(* Logix 5000 project; controller EsteiraSeletoraParte3 vendor 1 type 14 code 89 rev 20.11; software revision 20.05 *)

TASK MainTask (continuous, watchdog 500 ms) : MainProgram

MODULES
   Controller : vendor 1 type 14 code 89 (CompactLogixL23E_QBFC1_Controller 0, rev 20.11)
      LocalENB : vendor 1 type 12 code 191 (CompactLogixL23E_QBFC1_Ethernet 1, rev 20.11)
      Local : CompactBus (CompactVirtualAdapter 3, rev 20.11)
         Discrete_Inputs : vendor 1 type 7 code 320 (Compact 1, rev 3.1, Input RPI 20 ms)
         Discrete_Outputs : vendor 1 type 7 code 322 (Compact 2, rev 3.1, Output RPI 20 ms)
         Analog_IO : vendor 1 type 10 code 120 (Compact 3, rev 1.1, Output RPI 80 ms)
         Counters : vendor 1 type 109 code 70 (Compact 4, rev 1.1, Output RPI 20 ms)
END_MODULES

PROGRAM MainProgram   (* main routine MainRoutine *)
VAR
   AcionaEstacao1 : BOOL;
   AcionaEstacao2 : BOOL;
   AcionaEstacao3 : BOOL;
   EntroEstacao1 : BOOL;
   EntroEstacao2 : BOOL;
   EntroEstacao3 : BOOL;
   EsperaParaParar : TIMER;
   Estacao1 : BOOL;
   Estacao2 : BOOL;
   Estacao3 : BOOL;
   MotorEsteira : ALIAS FOR Local:2:O.Data.9;
   SensorEstacao1 : ALIAS FOR Local:1:I.Data.8;
   SensorEstacao2 : ALIAS FOR Local:1:I.Data.9;
   SensorEstacao3 : ALIAS FOR Local:1:I.Data.10;
   SistemaLigado : BOOL;
   StartStop : ALIAS FOR Local:1:I.Data.3;
   TrabalhandoEm1 : TIMER := (PRE := 1000);
   TrabalhandoEm2 : TIMER := (PRE := 2000);
   TrabalhandoEm3 : TIMER := (PRE := 3000);
END_VAR

ROUTINE MainRoutine   (* ladder *)
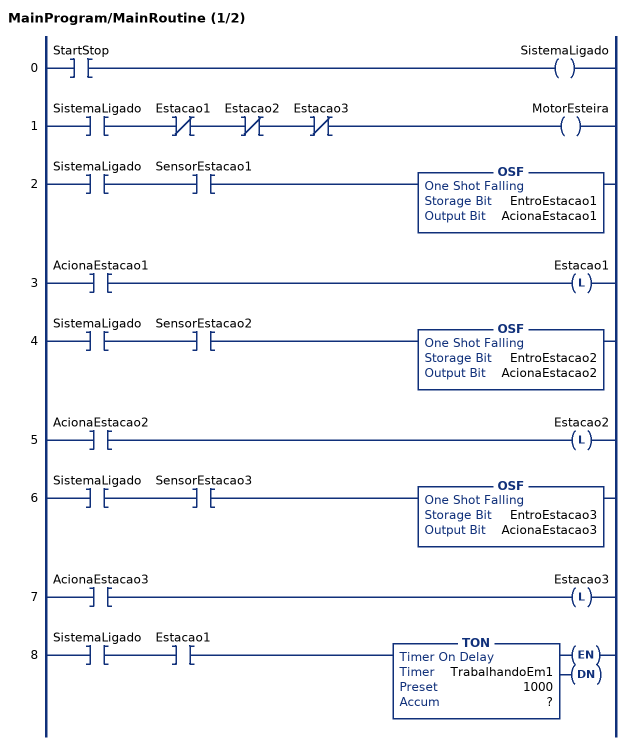
   0: XIC(StartStop)OTE(SistemaLigado);
   1: XIC(SistemaLigado)XIO(Estacao1)XIO(Estacao2)XIO(Estacao3)OTE(MotorEsteira);
   2: XIC(SistemaLigado)XIC(SensorEstacao1)OSF(EntroEstacao1,AcionaEstacao1);
   3: XIC(AcionaEstacao1)OTL(Estacao1);
   4: XIC(SistemaLigado)XIC(SensorEstacao2)OSF(EntroEstacao2,AcionaEstacao2);
   5: XIC(AcionaEstacao2)OTL(Estacao2);
   6: XIC(SistemaLigado)XIC(SensorEstacao3)OSF(EntroEstacao3,AcionaEstacao3);
   7: XIC(AcionaEstacao3)OTL(Estacao3);
   8: XIC(SistemaLigado)XIC(Estacao1)TON(TrabalhandoEm1,?,?);
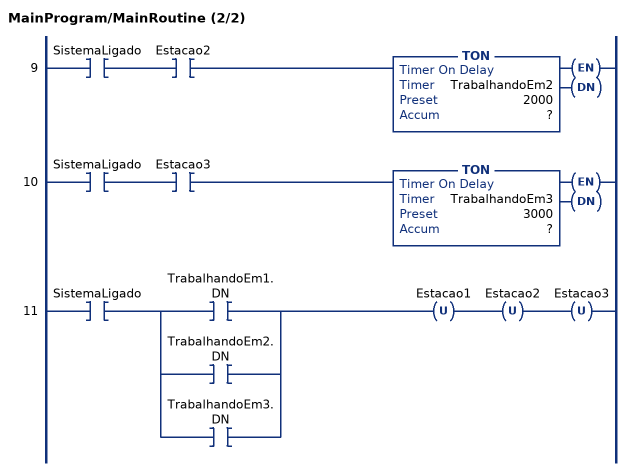
   9: XIC(SistemaLigado)XIC(Estacao2)TON(TrabalhandoEm2,?,?);
   10: XIC(SistemaLigado)XIC(Estacao3)TON(TrabalhandoEm3,?,?);
   11: XIC(SistemaLigado)[XIC(TrabalhandoEm1.DN) ,XIC(TrabalhandoEm2.DN) ,XIC(TrabalhandoEm3.DN) ]OTU(Estacao1)OTU(Estacao2)OTU(Estacao3);
END_ROUTINE
END_PROGRAM
